// TIA Portal V16 export
// export: Created 2024-12-03T15:41:40.7984089Z, ExportSetting WithDefaults, DisplayName Totally Integrated Automation Portal, DisplayVersion V16 Update 6, DisplayName TIA Portal Version Control Interface, DisplayVersion V16 Update 2, DisplayName TIA Portal Openness, DisplayVersion V16 Update 6, DisplayName TIA Portal Teamcenter Gateway, DisplayVersion V16, DisplayName SINAMICS Startdrive Advanced, DisplayVersion V16 Update 5, DisplayName SINAMICS Startdrive G130, G150, S120, S150, SINAMICS MV, S210, DisplayVersion V16 Update 5, DisplayName SINAMICS Startdrive G110M, G120, G120C, G120D, G120P, G115D, DisplayVersion V16 Update 5, DisplayName STEP 7 Professional, DisplayVersion V16 Update 6, DisplayName STEP 7 Safety, DisplayVersion V16, DisplayName WinCC Advanced / Unified PC, DisplayVersion V16 Update 6
FUNCTION_BLOCK "AlarmMain"   // FB43, SCL
{ S7_Optimized_Access := 'FALSE' }
VERSION : 0.1
// stored: AutoNumber true, IsIECCheckEnabled false, SetENOAutomatically false, UDAEnableTagReadback false
   VAR
      EMG_MAIN : "EMG_STATUS_FB";
      EMG_ZONE_1 { S7_SetPoint := 'True'} : "EMG_STATUS_FB";
      EMG_ZONE_2 { S7_SetPoint := 'True'} : "EMG_STATUS_FB";
      EMG_ZONE_3_4 { S7_SetPoint := 'True'} : "EMG_STATUS_FB";
      EMG_ZONE_5 : "EMG_STATUS_FB";
      DataCollectorConnection { S7_SetPoint := 'True'} : "ConnectionChecker_FB";
      Cmb24VNOK_1 { S7_SetPoint := 'True'} : Program_Alarm;
   END_VAR
   VAR_TEMP
      T_Condition : Bool;
   END_VAR
BEGIN
   REGION EMG MAIN NOK

       #T_Condition :=
       "I_EMG_MAIN" AND "I_EMG_ZONE_5B" AND
       "I_EMG_ZONE_2A" AND
       "I_EMG_ZONE_2B" AND
       "I_EMG_ZONE_3_4" AND
       "I_EMG_ZONE_5";

       #EMG_MAIN(I_BTTN_STATUS_OK := #T_Condition,
                 I_EMG_ACTIVATED := "I_EMG_MAIN",
                 I_UseEmgNotActiveAlarm := TRUE,
                 I_UseBttnPressedALarm := TRUE,
                 I_EmgName := 'EMG MAIN',
                 IO_STATUS := "EMG_STATUS_DB".EMG_MAIN);

   END_REGION

   REGION EMG MAIN ZONES

       #EMG_ZONE_1(I_BTTN_STATUS_OK := "I_EMG_ZONE_5B" OR TRUE,
                   I_EMG_ACTIVATED := FALSE,
                   I_UseEmgNotActiveAlarm := FALSE,
                   I_EmgName := 'EMG ZONE 1',
                   IO_STATUS := "EMG_STATUS_DB".EMG_ZONE_1);

       #EMG_ZONE_2(I_BTTN_STATUS_OK := "I_EMG_ZONE_2A" AND "I_EMG_ZONE_2B",
                   I_EMG_ACTIVATED := FALSE,
                   I_UseEmgNotActiveAlarm := FALSE,
                   I_EmgName := 'EMG ZONE 2',
                   IO_STATUS := "EMG_STATUS_DB".EMG_ZONE_2);

       #EMG_ZONE_3_4(I_BTTN_STATUS_OK := "I_EMG_ZONE_3_4",
                     I_EMG_ACTIVATED := FALSE,
                     I_UseEmgNotActiveAlarm := FALSE,
                     I_EmgName := 'EMG ZONE 3, ZONE 4',
                     IO_STATUS := "EMG_STATUS_DB".EMG_ZONE_3_4);

       #EMG_ZONE_5(I_BTTN_STATUS_OK := "I_EMG_ZONE_5" AND "I_EMG_ZONE_5B",
                   I_EMG_ACTIVATED := FALSE,
                   I_UseEmgNotActiveAlarm := FALSE,
                   I_EmgName := 'EMG ZONE 5',
                   IO_STATUS := "EMG_STATUS_DB".EMG_ZONE_5);

   END_REGION

   REGION 24V OK

       #Cmb24VNOK_1(SIG := NOT "I_EMG_MAIN" OR NOT "I_EMG_ZONE_5B");

   END_REGION


   REGION Alarm actvie shared

       "Alarms_DB".AlarmActiveShared :=
       #DataCollectorConnection.O_alarmActive OR
       #EMG_MAIN.O_AlarmActive OR
       "Alarms_DB".IPC_NotConnected;

   END_REGION

   REGION Alarm active

       "Alarms_DB".AlarmActive := "Alarms_DB".AlarmActiveShared;

   END_REGION
END_FUNCTION_BLOCK
